FUNCTION_BLOCK FB_SsNcConveyer IMPLEMENTS I_NcConveyer
VAR_INPUT
END_VAR
VAR_OUTPUT
END_VAR
VAR
	_Axis1	: AXIS_REF;
	_Axis2	: AXIS_REF;
	
END_VAR


PROPERTY Axis1 : Tc2_MC2.AXIS_REF
GET
Axis1 := _Axis1;
END_GET
SET
_Axis1 := Axis1;
END_SET
END_PROPERTY

PROPERTY Axis2 : Tc2_MC2.AXIS_REF
GET
Axis2 := _Axis2;
END_GET
SET
_Axis2 := Axis2;
END_SET
END_PROPERTY

METHOD Execute : BOOL
ADSLOGSTR(ADSLOG_MSGTYPE_LOG,'Moving short-straight','');
END_METHOD


METHOD Reset : BOOL
ADSLOGSTR(ADSLOG_MSGTYPE_LOG,'Reseting short-straight','');
END_METHOD

METHOD Start : BOOL
ADSLOGSTR(ADSLOG_MSGTYPE_LOG,'Powering Short-Straight on','');
END_METHOD

METHOD Stop : BOOL
ADSLOGSTR(ADSLOG_MSGTYPE_LOG,'Stopping short-straight','');
END_METHOD

END_FUNCTION_BLOCK

(* stored: Version 1.1.0.1, ProductVersion 3.1.4024.11
   POU FB_SsNcConveyer: Id {5570e42e-7ebf-4c22-865f-666c9a6f8ba2}, SpecialFunc None
   Property Axis1: Id {46e1d492-b2fe-4510-b67a-6641f6ec1782}
   Get Get: Id {1d681339-1217-4bea-aef1-8609a0d655ec}
   Set Set: Id {1c90a63f-3886-4bc2-99a5-5ee97c55af16}
   Property Axis2: Id {6ecdcf21-1cdf-46e4-8949-476a2563d481}
   Get Get: Id {f7e9ffa1-dc79-4ccf-b122-b3213bc6f894}
   Set Set: Id {dd21ffdb-2112-4bed-a09c-1f355e7ad169}
   Method Execute: Id {1db5a845-0ad9-4c13-bac5-eb33a1e9d23c}
   Method Reset: Id {50267c05-81d4-4041-a35c-bbb42bb35d43}
   Method Start: Id {99a1e3d0-bf7d-4fcd-aa1b-a42d40086359}
   Method Stop: Id {83e93853-423e-49f5-ba6f-fc72c2765a82} *)
